FUNCTION_BLOCK FB_OutRobot_BoxMoveReverse_Old EXTENDS FB_ObjectBase_V2
VAR_INPUT
//    Execute    :BOOL;   // True : This prog will start.
//    Abort      :BOOL;   // True : This prog will be abort.
//    Reset      :BOOL;   // True : This prog will be reset.
//    ObjectName :STRING; // Set this fb name(About it's action)
	INPUT            			   : REFERENCE TO ST_InputTable;
	Cylinder   					   : REFERENCE TO UNI_CylinderList;
	Motor      					   : REFERENCE TO UNI_MotorList;
	Cylinders					   : REFERENCE TO ARRAY[0..1] OF FB_Cylinder;
	Clips						   : REFERENCE TO ARRAY[0..1] OF FB_Cylinder;
	AutoMode_OutRobotMoveMove : st_AutoMode_ClampingBoxesJob;	
END_VAR

VAR_OUTPUT
//    Busy    :BOOL;        // True : This prog is running.
//    Done    :BOOL;        // True : Command has been executed.
//    Aborted :BOOL;        // True : This prog is aborted.
//    Error   :BOOL;        // True : This prog has an error.
//    ErrorID :UINT;       // Output ErrorID
//    Status  :T_MaxString; // Output this prog status by string(255bytes)
END_VAR

VAR
//    eState :E_MethodStatus_Basic;
//	uiExecutingStep : UDINT; // This var is used to been controll STATE_EXECUTING process.
//	uiResettingStep : UDINT;
//	uiAbortingStep : UDINT;
//	_Executed :BOOL; // Executing process completed.
//	_Error : BOOL; // FB has an error.
//	_ResetCompleted : BOOL; // FB resetting completed.
//	_AbortCompleted : BOOL; // FB aborting completed.
	//_Abort		: BOOL;
	strStatus	: STRING;
	uiResumeStep : UINT;
	tonTimeOut   :TON;
	tonTimeDelay   :TON;
	iWorkingIndex : INT;
	_UniqueErrorCode :STRING;
	
	
	PickingPos	: ARRAY[0..1] OF ST_PositionTable;
	PlacingPos  : ARRAY[0..1] OF ST_PositionTable;
	bSyncPick	: BOOL;
	bSyncPlace	: BOOL;
	SensorOnConveyor			   : BIT;
	ConveyorMotor				   : REFERENCE TO FB_Motor;
	UseA	: BOOL;
	UseB	: BOOL;
	bMotorMoveForward : BOOL;
END_VAR

A00_BasicUnits();
SUPER^.A10_StateControl();

ACTION A00_BasicUnits:
tonTimeOut(PT:=T#60S);
tonTimeDelay(PT:=T#1.5s);
END_ACTION

METHOD GetModelState
VAR_OUTPUT
    xDone    :BOOL;
    xBusy    :BOOL;
    xError   :BOOL;
    xAborted :BOOL;
    iErrorID :UDINT;
	UniqueErrorCode : STRING;
END_VAR
xDone    := Done;
xBusy    := Busy;
xError   := Error;
xAborted := Abort;
iErrorID := ErrorID;
UniqueErrorCode := THIS^.UniqueErrorCode;
END_METHOD

METHOD GetName : STRING
GetName := ObjectName;
END_METHOD

METHOD PRIVATE M_CheckCommand : BOOL
VAR_INPUT
END_VAR


M_CheckCommand:=true;
END_METHOD

METHOD PRIVATE M_GetWorkingConditions : BOOL
VAR_INPUT
END_VAR
//For Outbox move reverse, Boxes must place on same position , therefor only work with TargetPosition of ClipA

IF AutoMode_OutRobotMoveMove.ClampingInfo.TargetOfClipA = 5 THEN
	ConveyorMotor REF= Motor.List.TransmitDifferentSideCV;
ELSIF AutoMode_OutRobotMoveMove.ClampingInfo.TargetOfClipA = 6 THEN
	ConveyorMotor REF= Motor.List.TransmitSameSideCV;
ELSIF AutoMode_OutRobotMoveMove.ClampingInfo.TargetOfClipA = 3 THEN
	ConveyorMotor REF= Motor.List.TransmitDifferentSideCV;
ELSIF AutoMode_OutRobotMoveMove.ClampingInfo.TargetOfClipA = 4 THEN
	ConveyorMotor REF= Motor.List.TransmitSameSideCV;	
END_IF

IF AutoMode_OutRobotMoveMove.ClampingInfo.TargetOfClipA=5 THEN
		bMotorMoveForward := FALSE;
	ELSE
		bMotorMoveForward := TRUE;	
END_IF
IF AutoMode_OutRobotMoveMove.ClampingInfo.UseClibA THEN
	PickingPos[0] :=FUN_GetPositionTableData('R',1,0);
	UseA := TRUE;
	CASE  AutoMode_OutRobotMoveMove.ClampingInfo.TargetOfClipA OF	
		
	3,4:
		PlacingPos[0] :=FUN_GetPositionTableData('O',AutoMode_OutRobotMoveMove.ClampingInfo.TargetOfClipA,0);
	5,6:
		PlacingPos[0] :=FUN_GetPositionTableData('I',AutoMode_OutRobotMoveMove.ClampingInfo.TargetOfClipA,0);
	ELSE
		strStatus :='FB_OutRobot_BoxMoveReverse: Wrong command: Clip A target not allow';
		M_GetWorkingConditions := FALSE;
		RETURN;
	END_CASE
END_IF

IF AutoMode_OutRobotMoveMove.ClampingInfo.UseClibB THEN
	PickingPos[1] :=FUN_GetPositionTableData('R',2,1);
	UseB :=TRUE;
		CASE AutoMode_OutRobotMoveMove.ClampingInfo.TargetOfClipA OF
		
	3,4:
		PlacingPos[1] :=FUN_GetPositionTableData('O',AutoMode_OutRobotMoveMove.ClampingInfo.TargetOfClipA,1);
	5,6 :
		PlacingPos[1] :=FUN_GetPositionTableData('I',AutoMode_OutRobotMoveMove.ClampingInfo.TargetOfClipA,1);
	ELSE
		strStatus :='FB_OutRobot_BoxMoveReverse: Wrong command: Clip B target not allow';
		M_GetWorkingConditions := FALSE;
		RETURN;
	END_CASE
END_IF
IF PlacingPos[0].X_Pos =PlacingPos[1].X_Pos AND PlacingPos[0].Y_Pos = PlacingPos[1].Y_Pos AND UseA AND UseB THEN
		bSyncPlace:=TRUE;
	ELSE
		bSyncPlace:=FALSE;	
END_IF
IF PickingPos[0].X_Pos =PickingPos[1].X_Pos AND PickingPos[0].Y_Pos = PickingPos[1].Y_Pos AND UseA AND UseB THEN
		bSyncPick:=TRUE;
	ELSE
		bSyncPick:=FALSE;	
END_IF

M_GetWorkingConditions :=TRUE;
END_METHOD

METHOD PRIVATE M_RecoveryAllObjects : BOOL
VAR_INPUT
END_VAR
VAR 
	i : INT;
END_VAR
FOR i:=0 TO 1 DO
	IF Clips[i].xError THEN
		Clips[i].M_Reset();
		ELSE
		Clips[i].M_Retract();		
	END_IF
	IF Cylinders[i].xError THEN
	Cylinders[i].M_Reset();	
	ELSE
	Cylinders[i].M_Retract();	
	END_IF
END_FOR


IF arAxisCtrl_gb[AxisNo.OutRobot_X].Admin.Axis.Status.Error THEN

	arAxisCtrl_gb[AxisNo.OutRobot_X].Admin.ClearError:= TRUE;
ELSE
	arAxisCtrl_gb[AxisNo.OutRobot_X].Admin.ClearError:= FALSE;
END_IF

IF arAxisCtrl_gb[AxisNo.OutRobot_Y].Admin.Axis.Status.Error THEN

	arAxisCtrl_gb[AxisNo.OutRobot_Y].Admin.ClearError:= TRUE;
ELSE
	arAxisCtrl_gb[AxisNo.OutRobot_Y].Admin.ClearError:= FALSE;
END_IF
END_METHOD

METHOD PRIVATE M_SensorUpdate : BOOL
VAR_INPUT
END_VAR
IF AutoMode_OutRobotMoveMove.ClampingInfo.TargetOfClipA = 5 THEN
	SensorOnConveyor := INPUT.bDifferentSizeCV_BoxDetect5_Sensor;
ELSIF AutoMode_OutRobotMoveMove.ClampingInfo.TargetOfClipA = 6 THEN
	SensorOnConveyor := INPUT.bSameSizeCV_BoxDetect5_Sensor;
ELSIF AutoMode_OutRobotMoveMove.ClampingInfo.TargetOfClipA = 3 THEN
	SensorOnConveyor := INPUT.bDifferentSizeCV_BoxDetect4_Sensor;
ELSIF AutoMode_OutRobotMoveMove.ClampingInfo.TargetOfClipA = 4 THEN
	SensorOnConveyor := INPUT.bSameSizeCV_BoxDetect4_Sensor;	
END_IF
END_METHOD

METHOD  M_STATE_ABORTED
VAR_INPUT
END_VAR
ERROR :=TRUE;
Busy    := FALSE;
Aborted := TRUE;
Status := strStatus;

IF NOT Execute THEN
	eSTATE:=STATE_RESETTING;
END_IF

IF Execute AND Reset THEN
//	uiExecutingStep :=uiResumeStep;
	eSTATE:=STATE_EXECUTING;
END_IF
END_METHOD

METHOD  M_STATE_ABORTING
VAR_INPUT
END_VAR

VAR
	i : int;
	bCylinderCheck: BOOL;
END_VAR
Error :=True;
CASE uiAbortingStep OF
	0 :
		bCylinderCheck:=TRUE;
		ConveyorMotor.M_MotorStop();
		FOR i :=0 TO 1 DO		
	    	Cylinders[i].M_Reset();
			Cylinders[i].M_Retract();
			bCylinderCheck:=bCylinderCheck AND Cylinders[i].InRearPosition;	
		END_FOR
		IF bCylinderCheck THEN		
			uiAbortingStep:=9999;
		END_IF
		
	9999:	
			_AbortCompleted:=TRUE;
END_CASE

IF _AbortCompleted THEN	
	eSTATE :=STATE_ABORTED;
END_IF
END_METHOD

METHOD  M_STATE_DONE
VAR_INPUT
END_VAR
Busy 	:= FALSE;
Done	:=TRUE;

IF NOT Execute THEN
	eSTATE:=STATE_RESETTING;
END_IF
END_METHOD

METHOD  M_STATE_DORMANT
VAR_INPUT
END_VAR
Busy            := FALSE;
Done            := FALSE;
Aborted         := FALSE;
Error           := FALSE;
ErrorID         := 0;
Status          := '';
_ResetCompleted := FALSE;
_Error          := FALSE;
_Executed       := FALSE;
strStatus :='FB_OutRobot_BoxMoveReverse: No Error';
uiExecutingStep :=uiResettingStep :=uiResumeStep :=0;
tonTimeOut.IN :=TRUE;
_UniqueErrorCode:='0';
iWorkingIndex :=0;
bSyncPick :=FALSE;
bSyncPlace := FALSE;
UseA := FALSE;
UseB :=FALSE;
bMotorMoveForward:= FALSE;

IF Execute THEN
	eSTATE:=STATE_EXECUTING;
END_IF
END_METHOD

METHOD  M_STATE_ERROR
VAR_INPUT
END_VAR
ERROR   :=TRUE;
Busy	:=FALSE;
Status := strStatus;
ConveyorMotor.M_MotorStop();

IF NOT Execute THEN	
eSTATE:=STATE_RESETTING;
END_IF
END_METHOD

METHOD  M_STATE_EXECUTING
VAR_INPUT
END_VAR
VAR_INST
	bMoveConveyorForward : BOOL;
	bMoveConveyorBackrward : bool;
END_VAR

VAR
	bCylinderCheck : BOOL := TRUE;
END_VAR
Busy :=TRUE;
M_SensorUpdate();
IF bMoveConveyorForward THEN
	IF NOT ConveyorMotor.InBackWard THEN
		ConveyorMotor.M_MoveForward();	
	END_IF
END_IF

IF bMoveConveyorBackrward THEN
	IF NOT ConveyorMotor.InForWard THEN
		ConveyorMotor.M_MoveBackward();
	END_IF
END_IF
CASE uiExecutingStep OF
	

0: //Idle
bMoveConveyorForward:=FALSE;
bMoveConveyorBackrward:=FALSE;
	tonTimeDelay.IN :=FALSE;
	tonTimeOut.IN := FALSE;
	M_RecoveryAllObjects();
	//M_GetWorkingConditions();
	iWorkingIndex :=0;
	uiExecutingStep := 100;
	
100: //Check command
	IF M_GetWorkingConditions()THEN
		uiExecutingStep:=200;
	ELSE
		_Error:=TRUE;		
	END_IF
	
200: // first index

		IF UseA THEN
			iWorkingIndex :=0;
		ELSE
			iWorkingIndex :=1;	
		END_IF
		
		uiExecutingStep:=1000;	
	
1000: 
	// Move OutRobot to First clip picking	
	 	 
	arAxisCtrl_gb[AxisNo.OutRobot_X].PosMode.Position := PickingPos[iWorkingIndex].X_Pos;		
	arAxisCtrl_gb[AxisNo.OutRobot_Y].PosMode.Position := PickingPos[iWorkingIndex].Y_Pos;	
	uiExecutingStep:=1100;
		// todo : Check axes is moving
1100:
	// Check outRobot arrived
	IF		(arAxisStatus_gb[AxisNo.OutRobot_X].Admin._OpModeAck = ModePosAbs AND arAxisStatus_gb[AxisNo.OutRobot_X].Admin.CmdDone) 
	AND (arAxisStatus_gb[AxisNo.OutRobot_Y].Admin._OpModeAck = ModePosAbs AND arAxisStatus_gb[AxisNo.OutRobot_Y].Admin.CmdDone) 
	THEN
		tonTimeOut.IN := FALSE;
		uiExecutingStep:=1200;
	END_IF	
	tonTimeOut.IN := TRUE;
	IF tonTimeOut.q THEN
		tonTimeOut.IN := FALSE;
		_Error := TRUE;
		strStatus :='FB_OutRobot_BoxMoveReverse Step 1100: Move Robot to picking position timeout';
	END_IF
1200: //Clip Down Pick	  
	bCylinderCheck := TRUE;
	Cylinders[iWorkingIndex].M_Extend();
	bCylinderCheck := Cylinders[iWorkingIndex].InFrontPosition AND bCylinderCheck;
	IF bSyncPick THEN
		Cylinders[1].M_Extend();
		bCylinderCheck := Cylinders[1].InFrontPosition AND bCylinderCheck;
	END_IF	
	 
	IF bCylinderCheck THEN
		tonTimeOut.IN := FALSE;
		uiExecutingStep:=1300;
	END_IF 
	tonTimeOut.IN := TRUE;
	IF tonTimeOut.q THEN
		tonTimeOut.IN := FALSE;
		_Abort := TRUE;
		strStatus :='FB_OutRobot_BoxMoveReverse Step 1200: Cylinder pick down timeout';
	END_IF
	
1300: // Clip close Pick
	bCylinderCheck := TRUE;
	Clips[iWorkingIndex].M_Extend();
	bCylinderCheck := Clips[iWorkingIndex].InFrontPosition AND bCylinderCheck;
	IF bSyncPick THEN
		Clips[1].M_Extend();
		bCylinderCheck := Clips[1].InFrontPosition AND bCylinderCheck;
	END_IF	
	 
	IF bCylinderCheck THEN
		tonTimeOut.IN := FALSE;
		uiExecutingStep:=1400;
	END_IF 
	tonTimeOut.IN := TRUE;
	IF tonTimeOut.q THEN
		tonTimeOut.IN := FALSE;
		_Abort := TRUE;
		strStatus :='FB_OutRobot_BoxMoveReverse Step 1300: Clip pick close timeout';
	END_IF
	
1400: // Clip Up Pick
	bCylinderCheck := TRUE;
	Cylinders[iWorkingIndex].M_Retract();
	bCylinderCheck := Cylinders[iWorkingIndex].InRearPosition AND bCylinderCheck;
	IF bSyncPick THEN
		Cylinders[1].M_Retract();
		bCylinderCheck := Cylinders[1].InRearPosition AND bCylinderCheck;
	END_IF	
	 
	IF bCylinderCheck THEN
		tonTimeOut.IN := FALSE;
		uiExecutingStep:=1500;
	END_IF 
	  tonTimeOut.IN := TRUE;
	IF tonTimeOut.q THEN
		tonTimeOut.IN := FALSE;
		_Abort := TRUE;
		strStatus :='FB_OutRobot_BoxMoveReverse Step 1400: Cylinder pick up timeout';
	END_IF
	
1500: // If Next pick
	  IF iWorkingIndex>=1 OR bSyncPick OR NOT UseB THEN
		//Go to placing step
			IF UseA THEN
				iWorkingIndex:=0;
			ELSE
				iWorkingIndex:=1;	
			END_IF
			uiExecutingStep:=2000;
		ELSE
			iWorkingIndex :=iWorkingIndex +1;
			uiExecutingStep:=1000;	
	  END_IF
	  

2000: // Move to Placing pos
	  // Move Conveyor 
	   IF bMotorMoveForward THEN
		 	bMoveConveyorForward:=TRUE;//ConveyorMotor.M_MoveForward();
			bMoveConveyorBackrward := FALSE;
		  ELSE	 
			  bMoveConveyorForward := FALSE;
			 bMoveConveyorBackrward := TRUE; 
	 		 ConveyorMotor.M_MoveBackward(); 
	   END_IF
	   
	 arAxisCtrl_gb[AxisNo.OutRobot_X].PosMode.Position := PlacingPos[iWorkingIndex].X_Pos;		
	 arAxisCtrl_gb[AxisNo.OutRobot_Y].PosMode.Position := PlacingPos[iWorkingIndex].Y_Pos;	
	 uiExecutingStep:=2100;

2100: // Waiting outRobot move to placing pos	 
	  // Check sensor off for a while
	tonTimeDelay.IN := NOT 	SensorOnConveyor;
	 IF	(arAxisStatus_gb[AxisNo.OutRobot_X].Admin._OpModeAck = ModePosAbs AND arAxisStatus_gb[AxisNo.OutRobot_X].Admin.CmdDone) 
	AND (arAxisStatus_gb[AxisNo.OutRobot_Y].Admin._OpModeAck = ModePosAbs AND arAxisStatus_gb[AxisNo.OutRobot_Y].Admin.CmdDone)
	AND  tonTimeDelay.Q
	THEN	
		tonTimeOut.IN := FALSE;	
		uiExecutingStep:=2150;
	END_IF	
	
	  tonTimeOut.IN := TRUE;
	IF tonTimeOut.q THEN
		tonTimeOut.IN := FALSE;
		_Error := TRUE;
		strStatus :='FB_OutRobot_BoxMoveReverse Step 2100: Move Robot to placing position time out';
	END_IF
	
2150 : //Motor stop
		tonTimeDelay.IN := FALSE;
		bMoveConveyorForward:=FALSE;
		bMoveConveyorBackrward:=FALSE;
		ConveyorMotor.M_MotorStop();
		IF	ConveyorMotor.InStopped THEN
			uiExecutingStep:=2200;
		END_IF

2200: //Cllp Down place
	bCylinderCheck := TRUE;
	Cylinders[iWorkingIndex].M_Extend();
	bCylinderCheck := Cylinders[iWorkingIndex].InFrontPosition AND bCylinderCheck;
	IF bSyncPlace THEN
		Cylinders[1].M_Extend();
		bCylinderCheck := Cylinders[1].InFrontPosition AND bCylinderCheck;
	END_IF	
	 
	IF bCylinderCheck THEN
		tonTimeOut.IN := FALSE;
		uiExecutingStep:=2300;
	END_IF 
	
	  tonTimeOut.IN := TRUE;
	IF tonTimeOut.q THEN
		tonTimeOut.IN := FALSE;
		_Abort := TRUE;
		strStatus :='FB_OutRobot_BoxMoveReverse Step 2200: Cylinder place down timeout';
	END_IF
	
2300: // Clip open Place
	bCylinderCheck := TRUE;
	Clips[iWorkingIndex].M_Retract();
	bCylinderCheck := Clips[iWorkingIndex].InRearPosition AND bCylinderCheck;
	IF bSyncPlace THEN
		Clips[1].M_Retract();
		bCylinderCheck := Clips[1].InRearPosition AND bCylinderCheck;
	END_IF	
	 
	IF bCylinderCheck THEN
		tonTimeOut.IN := FALSE;
		uiExecutingStep:=2400;
	END_IF 
	 tonTimeOut.IN := TRUE;
	IF tonTimeOut.q THEN
		tonTimeOut.IN := FALSE;
		_Abort := TRUE;
		strStatus :='FB_OutRobot_BoxMoveReverse Step 2300: Clip place open timeout';
	END_IF  
	  
2400: // Clip up Placing
	bCylinderCheck := TRUE;
	Cylinders[iWorkingIndex].M_Retract();
	bCylinderCheck := Cylinders[iWorkingIndex].InRearPosition AND bCylinderCheck;
	IF bSyncPlace THEN
		Cylinders[1].M_Retract();
		bCylinderCheck := Cylinders[1].InRearPosition AND bCylinderCheck;
	END_IF	
	 
	IF bCylinderCheck THEN
		tonTimeOut.IN := FALSE;
		uiExecutingStep:=2500;
	END_IF 
	 tonTimeOut.IN := TRUE;
	IF tonTimeOut.q THEN
		tonTimeOut.IN := FALSE;
		_Abort := TRUE;
		strStatus :='FB_OutRobot_BoxMoveReverse Step 2400: Cylinder place up timeout';
	END_IF  
	
2500: // If Next place
	IF iWorkingIndex>=1 OR bSyncPlace OR NOT UseB THEN
		uiExecutingStep:=2600;
		// Finish
	ELSE	
		iWorkingIndex := iWorkingIndex+1;
	  	uiExecutingStep:=2000;
	END_IF

2600: // Move conveyor a bit
		  IF bMotorMoveForward THEN
			 bMoveConveyorForward:=TRUE;//ConveyorMotor.M_MoveForward();
			 bMoveConveyorBackrward:=FALSE;
		  ELSE	 
			  bMoveConveyorForward:=FALSE;
			  bMoveConveyorBackrward:=TRUE;
	 		 ConveyorMotor.M_MoveBackward(); 
		  END_IF
		tonTimeDelay.IN := NOT SensorOnConveyor;		
		IF tonTimeDelay.Q THEN
			uiExecutingStep:=2700;
		END_IF
2700: // Stop movor
		bMoveConveyorForward:=FALSE;
		bMoveConveyorBackrward:=FALSE;
		ConveyorMotor.M_MotorStop();
		tonTimeDelay.IN := FALSE;
		IF ConveyorMotor.InStopped THEN
			uiExecutingStep:=3000;
		END_IF
3000: // Finish	
	_Executed:=TRUE;
	
END_CASE
	
IF NOT Execute THEN
	eState:=STATE_RESETTING;
END_IF
IF _Error THEN
	eState:=STATE_ERROR;
END_IF
IF _Abort THEN
	eSTATE:=STATE_ABORTING;
END_IF
IF _Executed THEN
	eSTATE:=STATE_Done;
END_IF
END_METHOD

METHOD  M_STATE_RESETTING
VAR_INPUT
END_VAR
Error :=_Error;
Done :=_Executed;
Busy := FALSE;


CASE uiResettingStep OF
	
	0:
		ConveyorMotor.M_MotorStop();
		M_RecoveryAllObjects();
		uiResettingStep:=9999;


	9999:
		M_RecoveryAllObjects();
		_ResetCompleted:=TRUE;
END_CASE
IF _ResetCompleted THEN
	eSTATE:=STATE_DORMANT;
END_IF
END_METHOD

END_FUNCTION_BLOCK

(* stored: Version 1.1.0.1, ProductVersion 3.1.4024.13
   POU FB_OutRobot_BoxMoveReverse_Old: Id {2010a4e0-e6c4-4a61-ade6-1d88897847d3}, SpecialFunc None
   Folder Method: Id {3226158d-4665-4849-bf0c-83df847d8e4a}
   Folder STATE: Id {b81dde6d-c30a-4b4f-9274-d386d378fe4a}
   Action A00_BasicUnits: Id {871c1988-dc90-4a56-b253-eb8b77b8a4b4}
   Method GetModelState: Id {87d57486-748b-4b84-893f-708c478b8089}
   Method GetName: Id {d60fa25c-e3a4-4da5-8b54-f31985b997b8}
   Method M_CheckCommand: Id {99b0aba1-caca-4248-a190-29327f26fc04}
   Method M_GetWorkingConditions: Id {b1f356aa-a92c-41ce-8e7d-9ad847c21bd2}
   Method M_RecoveryAllObjects: Id {fc7678d4-bb65-45fd-862f-96a4a21c1b30}
   Method M_SensorUpdate: Id {621a30f3-02f4-40fd-897f-cf5bab1b722f}
   Method M_STATE_ABORTED: Id {c3c5ce99-5e57-43a4-827f-558adde51648}
   Method M_STATE_ABORTING: Id {cca0af9f-77a9-4f29-b0f8-60b0f27bb3c8}
   Method M_STATE_DONE: Id {d11bc627-b501-4bb8-a371-5ee132806827}
   Method M_STATE_DORMANT: Id {2411840d-d85f-41c9-82a8-f7ff09309fa8}
   Method M_STATE_ERROR: Id {7426c8a7-ac70-4583-98a7-d373e0b17bca}
   Method M_STATE_EXECUTING: Id {a4f8385a-88e7-4ec2-972c-1f67f72164d1}
   Method M_STATE_RESETTING: Id {6022a289-1bf1-4584-84c6-fbde58184ef2} *)
